Fanuc KAREL source: kt00178.KL

-- PROVISIONAL review KL for V940-1; original PC SHA256 df242866ec4b9393c2e3239b7f9b6371ea41cafea9854b7fabcd30a76141c03f
-- Incomplete behavior may be omitted. Consult companion uncertainty JSON. Do not deploy.
PROGRAM KT00178
%NOLOCKGROUP
VAR
  I2 : INTEGER
  OUT : REAL
-- UNRESOLVED_DECL Y1 type=002018
BEGIN
  -- V9_ZERO_TABLE_METADATA_HINT layout=0001; no indexed target words; source/name/runtime held
  -- UNRESOLVED_PC offsets 5-19; opcodes 2E,22,9D,33,B2
  -- UNRESOLVED_PC offsets 24-35; opcodes 2E,23
  -- UNRESOLVED_PC offsets 40-63; opcodes 22,9D,33,B1,21,56,64,23
  -- UNRESOLVED_PC offsets 68-72; opcodes 7F
END KT00178
